(* Logix 5000 project; controller EuniceF_ICA4 vendor 1 type 14 code 150 rev 37.11; software revision 37.00 *)

TASK MainTask (continuous, watchdog 500 ms) : MainProgram

MODULES
   Local : vendor 1 type 14 code 150 (Compact 0, rev 37.11)
      Discrete_IO : Embedded (Compact 1, rev 3.1, Output RPI 20 ms)
      Analog_IO : Embedded (Compact 2, rev 1.1, Output RPI 80 ms)
      Counters : Embedded (Compact 3, rev 1.1, Output RPI 20 ms)
END_MODULES

VAR_GLOBAL   (* controller tags *)
   LOCK : ALIAS FOR Local:1:O.Data.2;
   M : ALIAS FOR Local:1:O.Data.4;
   M1 : ALIAS FOR Local:1:O.Data.0;
   M2 : ALIAS FOR Local:1:O.Data.1;
   M3 : ALIAS FOR Local:1:O.Data.3;
   RSESET : ALIAS FOR Local:1:I.Data.13;
   START : ALIAS FOR Local:1:I.Data.11;
   START2 : ALIAS FOR Local:1:I.Data.12;
   STOP : ALIAS FOR Local:1:I.Data.10;
   STOP1 : ALIAS FOR Local:1:I.Data.8;
END_VAR

PROGRAM MainProgram   (* main routine MainRoutine *)

ROUTINE MainRoutine   (* ladder *)
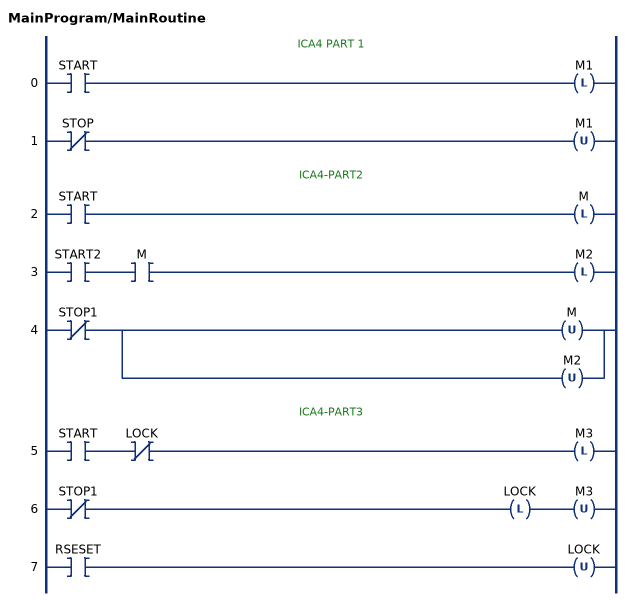
   // ICA4 PART 1
   0: XIC(START)OTL(M1);
   1: XIO(STOP)OTU(M1);
   // ICA4-PART2
   2: XIC(START)OTL(M);
   3: XIC(START2)XIC(M)OTL(M2);
   4: XIO(STOP1)[OTU(M) ,OTU(M2) ];
   // ICA4-PART3
   5: XIC(START)XIO(LOCK)OTL(M3);
   6: XIO(STOP1)OTL(LOCK)OTU(M3);
   7: XIC(RSESET)OTU(LOCK);
END_ROUTINE
END_PROGRAM
